Fanuc KAREL source: kx00010.KL

-- PROVISIONAL review KL for V770-1; original PC SHA256 7408c704e0147b9915ec3a8bd6c7da10326bb936a89cdf6f31fac9f410e0b76c
-- Incomplete behavior may be omitted. Consult companion uncertainty JSON. Do not deploy.
PROGRAM KX00010
%NOLOCKGROUP
VAR
  I : INTEGER
  J : INTEGER
  B : BOOLEAN
  F : FILE
  S : STRING[80]
-- UNRESOLVED_DECL P type=000102
BEGIN
  -- UNRESOLVED_PC offsets 5-7; opcodes 9C,10
  -- UNRESOLVED_PC offsets 12-16; opcodes 7F
END KX00010
